// TIA Portal V18 export
FUNCTION "SR1000" : Void   // FC1800, LAD
{ S7_Optimized_Access := 'TRUE' }
VERSION : 0.1
// stored: AutoNumber false, IsIECCheckEnabled false, SetENOAutomatically false, UDAEnableTagReadback false
BEGIN

REGION Network 1: 801A1
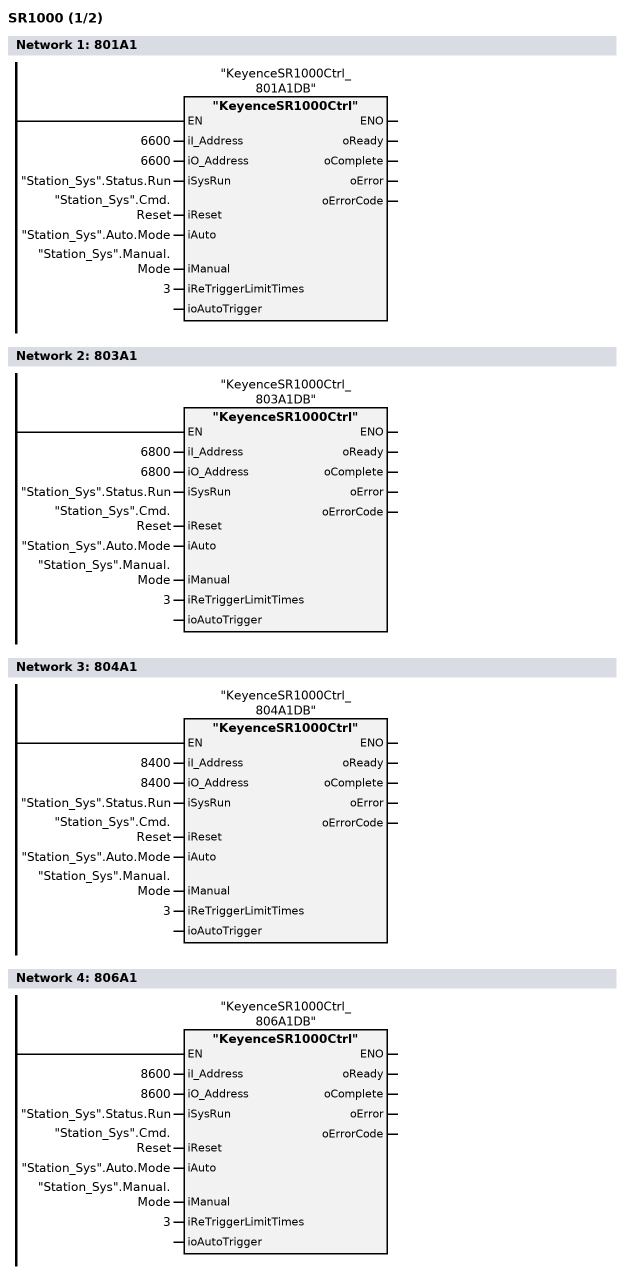
   RUNG wire#powerrail
      "KeyenceSR1000Ctrl_801A1DB"(iI_Address := 6600, iO_Address := 6600, iSysRun := "Station_Sys".Status.Run, iReset := "Station_Sys".Cmd.Reset, iAuto := "Station_Sys".Auto.Mode, iManual := "Station_Sys".Manual.Mode, iReTriggerLimitTimes := 3, ioAutoTrigger :=, oReady =>, oComplete =>, oError =>, oErrorCode =>)
   END_RUNG
   // the same network as SCL:
   "KeyenceSR1000Ctrl_801A1DB"(iI_Address := 6600,   // "KeyenceSR1000Ctrl"
                           iO_Address := 6600,
                           iSysRun := "Station_Sys".Status.Run,
                           iReset := "Station_Sys".Cmd.Reset,
                           iAuto := "Station_Sys".Auto.Mode,
                           iManual := "Station_Sys".Manual.Mode,
                           iReTriggerLimitTimes := 3);
END_REGION

REGION Network 2: 803A1
   RUNG wire#powerrail
      "KeyenceSR1000Ctrl_803A1DB"(iI_Address := 6800, iO_Address := 6800, iSysRun := "Station_Sys".Status.Run, iReset := "Station_Sys".Cmd.Reset, iAuto := "Station_Sys".Auto.Mode, iManual := "Station_Sys".Manual.Mode, iReTriggerLimitTimes := 3, ioAutoTrigger :=, oReady =>, oComplete =>, oError =>, oErrorCode =>)
   END_RUNG
   // the same network as SCL:
   "KeyenceSR1000Ctrl_803A1DB"(iI_Address := 6800,   // "KeyenceSR1000Ctrl"
                           iO_Address := 6800,
                           iSysRun := "Station_Sys".Status.Run,
                           iReset := "Station_Sys".Cmd.Reset,
                           iAuto := "Station_Sys".Auto.Mode,
                           iManual := "Station_Sys".Manual.Mode,
                           iReTriggerLimitTimes := 3);
END_REGION

REGION Network 3: 804A1
   RUNG wire#powerrail
      "KeyenceSR1000Ctrl_804A1DB"(iI_Address := 8400, iO_Address := 8400, iSysRun := "Station_Sys".Status.Run, iReset := "Station_Sys".Cmd.Reset, iAuto := "Station_Sys".Auto.Mode, iManual := "Station_Sys".Manual.Mode, iReTriggerLimitTimes := 3, ioAutoTrigger :=, oReady =>, oComplete =>, oError =>, oErrorCode =>)
   END_RUNG
   // the same network as SCL:
   "KeyenceSR1000Ctrl_804A1DB"(iI_Address := 8400,   // "KeyenceSR1000Ctrl"
                           iO_Address := 8400,
                           iSysRun := "Station_Sys".Status.Run,
                           iReset := "Station_Sys".Cmd.Reset,
                           iAuto := "Station_Sys".Auto.Mode,
                           iManual := "Station_Sys".Manual.Mode,
                           iReTriggerLimitTimes := 3);
END_REGION

REGION Network 4: 806A1
   RUNG wire#powerrail
      "KeyenceSR1000Ctrl_806A1DB"(iI_Address := 8600, iO_Address := 8600, iSysRun := "Station_Sys".Status.Run, iReset := "Station_Sys".Cmd.Reset, iAuto := "Station_Sys".Auto.Mode, iManual := "Station_Sys".Manual.Mode, iReTriggerLimitTimes := 3, ioAutoTrigger :=, oReady =>, oComplete =>, oError =>, oErrorCode =>)
   END_RUNG
   // the same network as SCL:
   "KeyenceSR1000Ctrl_806A1DB"(iI_Address := 8600,   // "KeyenceSR1000Ctrl"
                           iO_Address := 8600,
                           iSysRun := "Station_Sys".Status.Run,
                           iReset := "Station_Sys".Cmd.Reset,
                           iAuto := "Station_Sys".Auto.Mode,
                           iManual := "Station_Sys".Manual.Mode,
                           iReTriggerLimitTimes := 3);
END_REGION

REGION Network 5: 800A1
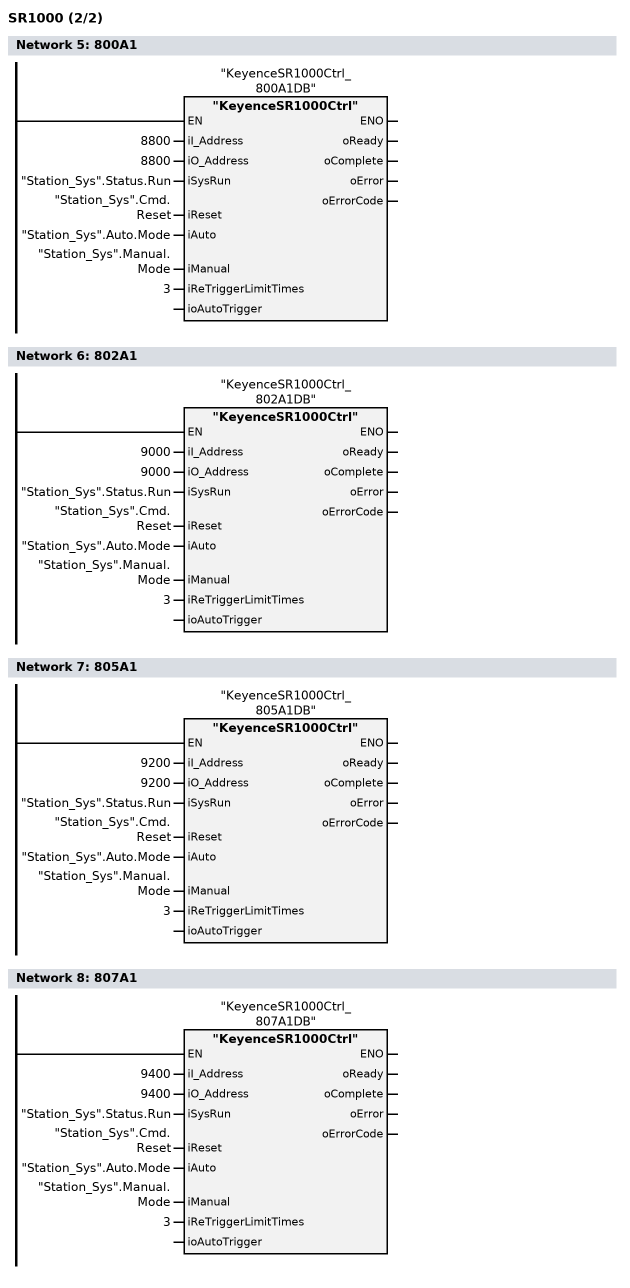
   RUNG wire#powerrail
      "KeyenceSR1000Ctrl_800A1DB"(iI_Address := 8800, iO_Address := 8800, iSysRun := "Station_Sys".Status.Run, iReset := "Station_Sys".Cmd.Reset, iAuto := "Station_Sys".Auto.Mode, iManual := "Station_Sys".Manual.Mode, iReTriggerLimitTimes := 3, ioAutoTrigger :=, oReady =>, oComplete =>, oError =>, oErrorCode =>)
   END_RUNG
   // the same network as SCL:
   "KeyenceSR1000Ctrl_800A1DB"(iI_Address := 8800,   // "KeyenceSR1000Ctrl"
                           iO_Address := 8800,
                           iSysRun := "Station_Sys".Status.Run,
                           iReset := "Station_Sys".Cmd.Reset,
                           iAuto := "Station_Sys".Auto.Mode,
                           iManual := "Station_Sys".Manual.Mode,
                           iReTriggerLimitTimes := 3);
END_REGION

REGION Network 6: 802A1
   RUNG wire#powerrail
      "KeyenceSR1000Ctrl_802A1DB"(iI_Address := 9000, iO_Address := 9000, iSysRun := "Station_Sys".Status.Run, iReset := "Station_Sys".Cmd.Reset, iAuto := "Station_Sys".Auto.Mode, iManual := "Station_Sys".Manual.Mode, iReTriggerLimitTimes := 3, ioAutoTrigger :=, oReady =>, oComplete =>, oError =>, oErrorCode =>)
   END_RUNG
   // the same network as SCL:
   "KeyenceSR1000Ctrl_802A1DB"(iI_Address := 9000,   // "KeyenceSR1000Ctrl"
                           iO_Address := 9000,
                           iSysRun := "Station_Sys".Status.Run,
                           iReset := "Station_Sys".Cmd.Reset,
                           iAuto := "Station_Sys".Auto.Mode,
                           iManual := "Station_Sys".Manual.Mode,
                           iReTriggerLimitTimes := 3);
END_REGION

REGION Network 7: 805A1
   RUNG wire#powerrail
      "KeyenceSR1000Ctrl_805A1DB"(iI_Address := 9200, iO_Address := 9200, iSysRun := "Station_Sys".Status.Run, iReset := "Station_Sys".Cmd.Reset, iAuto := "Station_Sys".Auto.Mode, iManual := "Station_Sys".Manual.Mode, iReTriggerLimitTimes := 3, ioAutoTrigger :=, oReady =>, oComplete =>, oError =>, oErrorCode =>)
   END_RUNG
   // the same network as SCL:
   "KeyenceSR1000Ctrl_805A1DB"(iI_Address := 9200,   // "KeyenceSR1000Ctrl"
                           iO_Address := 9200,
                           iSysRun := "Station_Sys".Status.Run,
                           iReset := "Station_Sys".Cmd.Reset,
                           iAuto := "Station_Sys".Auto.Mode,
                           iManual := "Station_Sys".Manual.Mode,
                           iReTriggerLimitTimes := 3);
END_REGION

REGION Network 8: 807A1
   RUNG wire#powerrail
      "KeyenceSR1000Ctrl_807A1DB"(iI_Address := 9400, iO_Address := 9400, iSysRun := "Station_Sys".Status.Run, iReset := "Station_Sys".Cmd.Reset, iAuto := "Station_Sys".Auto.Mode, iManual := "Station_Sys".Manual.Mode, iReTriggerLimitTimes := 3, ioAutoTrigger :=, oReady =>, oComplete =>, oError =>, oErrorCode =>)
   END_RUNG
   // the same network as SCL:
   "KeyenceSR1000Ctrl_807A1DB"(iI_Address := 9400,   // "KeyenceSR1000Ctrl"
                           iO_Address := 9400,
                           iSysRun := "Station_Sys".Status.Run,
                           iReset := "Station_Sys".Cmd.Reset,
                           iAuto := "Station_Sys".Auto.Mode,
                           iManual := "Station_Sys".Manual.Mode,
                           iReTriggerLimitTimes := 3);
END_REGION
END_FUNCTION
